(* IEC 61131-3 sources: ICSQuartz/benchmarks/oscat_basic_month_to_string/src, 1 file *)

(* ---- program.st ---- *)
PROGRAM PLC_PRG
VAR_INPUT
    in_MTH: INT;
    in_LANG: INT;
    in_LX: INT;
END_VAR

MONTH_TO_STRING(in_MTH, in_LANG, in_LX);

END_PROGRAM
